// TIA Portal project "cross_refences" (V18)

(* hardware
DEVICE "S7-1200 station_1"  S7-1200 Station
   slot 0: "Rack_0"  S7-1200 Rack  Rack  V1.0
   slot 1: "PLC_1"  CPU 1214C DC/DC/DC  6ES7 214-1AG40-0XB0  V4.6
*)

// ===== PLC "PLC_1"  CPU 1214C DC/DC/DC =====

FUNCTION "Tank_sicaklik_kontrolu" : Void   // FC1, LAD
{ S7_Optimized_Access := 'TRUE' }
VERSION : 0.1
   VAR_INPUT
      "SET DEĞERİ" : Bool;
      "GERÇEKLEŞEN DEĞER" : Bool;
      "HATA ORANI" : Bool;
      SICAKLIK : Bool;
   END_VAR
   VAR_OUTPUT
      ISITICI : Bool;
   END_VAR
BEGIN
END_FUNCTION

ORGANIZATION_BLOCK "Main"   // OB1, LAD, ProgramCycle
TITLE = "Main Program Sweep (Cycle)"
{ S7_Optimized_Access := 'TRUE' }
VERSION : 0.1
// PLcye sağ tıklayıp cross refence a erişim sağlayabiliriz ya da tools sekmesinden erişebiliriz.
   VAR_INPUT
      Initial_Call : Bool;   // Initial call of this OB
      Remanence : Bool;   // =True, if remanent data are available
   END_VAR
BEGIN

REGION Network 1
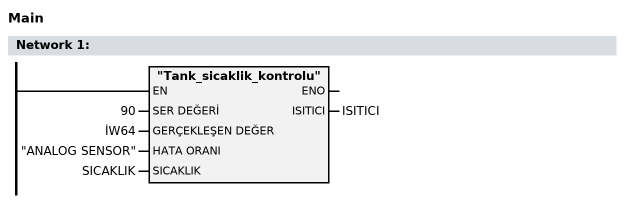
   RUNG wire#powerrail
      "Tank_sicaklik_kontrolu"("SER DEĞERİ" := 90, "GERÇEKLEŞEN DEĞER" := İW64, "HATA ORANI" := "ANALOG SENSOR", SICAKLIK := SICAKLIK, ISITICI => ISITICI)
   END_RUNG
   // the same network as SCL:
   "Tank_sicaklik_kontrolu"("SER DEĞERİ" := 90,
                           "GERÇEKLEŞEN DEĞER" := İW64,
                           "HATA ORANI" := "ANALOG SENSOR",
                           SICAKLIK := SICAKLIK,
                           ISITICI => ISITICI);
END_REGION
END_ORGANIZATION_BLOCK